// TIA Portal V16 export
// export: Created 2021-04-06T19:52:14.4941395Z, ExportSetting WithDefaults, DisplayName Totally Integrated Automation Portal, DisplayVersion V16, DisplayName TIA Portal Version Control Interface, DisplayVersion V16, DisplayName TIA Portal Openness, DisplayVersion V16, DisplayName STEP 7 Professional, DisplayVersion V16, DisplayName STEP 7 Safety, DisplayVersion V16, DisplayName WinCC Unified SCADA Engineering System, DisplayVersion V16
FUNCTION "pushToArray" : Void   // FC5, LAD
{ S7_Optimized_Access := 'TRUE' }
VERSION : 0.1
// stored: AutoNumber true, IsIECCheckEnabled false, SetENOAutomatically false, UDAEnableTagReadback false
   VAR_INPUT
      addValue : Real;
   END_VAR
   VAR_IN_OUT
      "array" : Array[*] of Real;
   END_VAR
   VAR_TEMP
      lowIndex : DInt;
      highIndex : DInt;
      i : SInt;
   END_VAR
BEGIN

REGION Network 1 (SCL)
   #lowIndex := LOWER_BOUND(ARR := #array, DIM := 1);
   #highIndex := UPPER_BOUND(ARR := #array, DIM := 1);

   #i := 0;
   FOR #i := (#highIndex - 1) TO #lowIndex BY -1 DO 
       #array[#i+1] := #array[#i];
   END_FOR;
   #array[#lowIndex] := #addValue;

   ENO := true;
END_REGION
END_FUNCTION
